// TIA Portal V19 export
DATA_BLOCK "Unit2Parameters"   // DB103
// stored: InstanceOfName LAF_typeHmiParameters, InstanceOfType UDT
"LAF_typeHmiParameters"
   // VAR
   //    em1 { S7_SetPoint := 'True'} : "LAF_typeRollerEm1ParametersHmi";
   //    em2 { S7_SetPoint := 'True'} : "LAF_typeConstraintRollerEm2ParametersHmi";
   //    em3 { S7_SetPoint := 'True'} : "LAF_typeConstraintWorkstationEm3ParametersHmi";
   //    em4 { S7_SetPoint := 'True'} : "LAF_typeXyzhandlingEm4ParametersHmi";
   //    em5 : "LAF_typePlasticWorkstationEm5ParametersHmi";
   //    em6 { S7_SetPoint := 'True'} : "LAF_typePlasticRollerEm6ParametersHmi";
   // END_VAR
BEGIN
   em1.cm1Vfd205.general.refSpeed := 1000.0;
   em1.cm1Vfd205.manual.upperVel := 500.0;
   em1.cm1Vfd205.manual.lowVel := 10.0;
   em1.cm1Vfd205.manual.highVel := 50.0;
   em1.cm1Vfd205.production.upperVel := 500.0;
   em1.cm1Vfd205.production.lowVel := 10.0;
   em1.cm1Vfd205.production.highVel := 50.0;
   em1.cm1Vfd205.maintenance.upperVel := 500.0;
   em1.cm1Vfd205.maintenance.lowVel := 10.0;
   em1.cm1Vfd205.maintenance.highVel := 50.0;
   em2.cm1Vfd206.manual.upperVel := 500.0;
   em2.cm1Vfd206.manual.lowVel := 10.0;
   em2.cm1Vfd206.manual.highVel := 50.0;
END_DATA_BLOCK
